{attribute 'qualified_only'}

//-----------------------------------------------------------------------------------------
//
//                  				GV_OpMode
//
//								Variables op Mode 			
//-----------------------------------------------------------------------------------------
//
//Auteur: G.GOETZ
//Création: 20.02.2026
//Dernière modification : 20.02.2026 (G.GOETZ)
//       			
//-----------------------------------------------------------------------------------------
//
//     							Liste des modifications  	
//
// 20.02.2026 (G.GOETZ) -> Création		
//-----------------------------------------------------------------------------------------

VAR_GLOBAL PERSISTENT
END_VAR

VAR_GLOBAL
	
	(** ENUM **)
		eOpModeRequest : ENUM_OpMode := ENUM_OpMode.None ;
		eOpMode : ENUM_OpMode := ENUM_OpMode.None ;

	(** PROCESS FLAG **)
		bInitAllowed : BOOL ; // Init is Allowed
		bAutoAllowed : BOOL ; // Auto is Allowed
		bManuAllowed : BOOL ; // Manu is Allowed

END_VAR

VAR_GLOBAL CONSTANT
END_VAR

(* stored: Version 1.1.0.1, ProductVersion 3.1.4026.17
   GVL GV_OpMode: Id {762ae7a7-776f-4e9f-afc6-9eda903018e6} *)
